FUNCTION Matrix_TransposeSquare : BOOL
VAR_INPUT
	M : REFERENCE TO Matrix;
END_VAR
VAR
	Ri : UINT;
	Ci : UINT;
	Temp : LREAL;
END_VAR

IF NOT(M.IsSquare) OR M.isempty THEN
	Matrix_TransposeSquare := FALSE;
	RETURN;
END_IF

Matrix_TransposeSquare := TRUE;

IF M.Length <= 1 THEN
	RETURN;
END_IF

FOR Ri := 0 TO M.Rows-2 DO
	FOR Ci := Ri+1 TO M.Cols-1 DO
		Temp := M.GetRC(Ri,Ci);
		M.SetRC(Ri,Ci,M.GetRC(Ci,Ri));
		M.SetRC(Ci,Ri,Temp);
	END_FOR
END_FOR

END_FUNCTION

(* stored: Version 1.1.0.1, ProductVersion 3.1.4024.9
   POU Matrix_TransposeSquare: Id {cddc94bc-80ef-0bdc-2507-33761c831052}, SpecialFunc None *)
